PROGRAM MAIN
VAR
	test: BOOL;
END_VAR

test := 1;

END_PROGRAM

(* stored: Version 1.1.0.1, ProductVersion 3.1.4024.10
   POU MAIN: Id {b2c178c7-064e-4039-923c-873a2e37011c}, SpecialFunc None *)
